{attribute 'linkalways'} 
{attribute 'no_explicit_call' := 'This FB is a CLASS and must be accessed using methods or properties'}
{attribute 'enable_dynamic_creation'}
FUNCTION_BLOCK FINAL Node_UDINT_TO_REAL EXTENDS Node
VAR
	in : _UDINT(0);
	out : _REAL(0.0);
	success : _BOOL(FALSE);
END_VAR

METHOD PUBLIC  Clone : I_Node
VAR
	pNode : POINTER TO Node_UDINT_TO_REAL;
END_VAR
pNode := __NEW(Node_UDINT_TO_REAL);
Clone := pNode^;
END_METHOD

METHOD FB_init : BOOL
VAR_INPUT
	bInitRetains : BOOL; // if TRUE, the retain variables are initialized (warm start / cold start)
	bInCopyCode : BOOL;  // if TRUE, the instance afterwards gets moved into the copy code (online change)
END_VAR
AddParameter('in', in);
AddOutput('out', out);
AddOutput('success', success);

this^.Metadatum.AddBoolAsMetadata('deprecated', true);
END_METHOD

METHOD PROTECTED OnExecute
VAR
END_VAR
success.Value := TryConvert_UDINT_TO_REAL(in.Value, out.Value);
END_METHOD

END_FUNCTION_BLOCK

(* stored: Version 1.1.0.1, ProductVersion 3.1.4026.18
   POU Node_UDINT_TO_REAL: Id {5bb88dd5-a25d-0276-2234-9f83e5cefd51}, SpecialFunc None
   Folder Constructor: Id {9bad18e9-3b54-0cf8-0522-9aa2842a0d8a}
   Method Clone: Id {a3ba2293-0d7e-0b39-17dd-d40a84957ff5}
   Method FB_init: Id {10e7587b-847f-04b6-3574-cc7fd8a1d5fe}
   Method OnExecute: Id {42c2cd12-f6b0-0b73-0bc5-e80f1aed40d7} *)
